TYPE AX5000_P_0601 :
STRUCT
	Predictive_velocity_command_value:DINT;
END_STRUCT
END_TYPE

(* stored: Version 1.1.0.1, ProductVersion 3.1.4024.3
   DUT AX5000_P_0601: Id {1cda4499-faad-4b4d-b913-189756b584cc} *)
